Staubli VAL3: motionStatus.pgx

public program motionStatus(num x_nInConnFlag)
begin

  // update connection status on port 11000 (motion server)

  gotoxy(scMonitor, 0,0)
  // 11 characteres: gotoxy(12,0) to insert status
  put(scMonitor, "Port 11000:")
  gotoxy(scMonitor, 12,0)
  switch x_nInConnFlag
    case -1
      put(scMonitor, "connection lost")
    break
    case 0
      put(scMonitor, "not connected")
    break
    case 1
      put(scMonitor, "connected")
    break
    default
      put(scMonitor, "not connected")
    break
  endSwitch

end
